// TIA Portal V19 export
FUNCTION "ALARMS" : Void   // FC16, LAD
{ S7_Optimized_Access := 'TRUE' }
// stored: SetENOAutomatically false
   VAR_TEMP   // added for the SCL form of the ladder/FBD networks
      _w1 : Bool;
   END_VAR
BEGIN

REGION Network 1: EMG ALARM
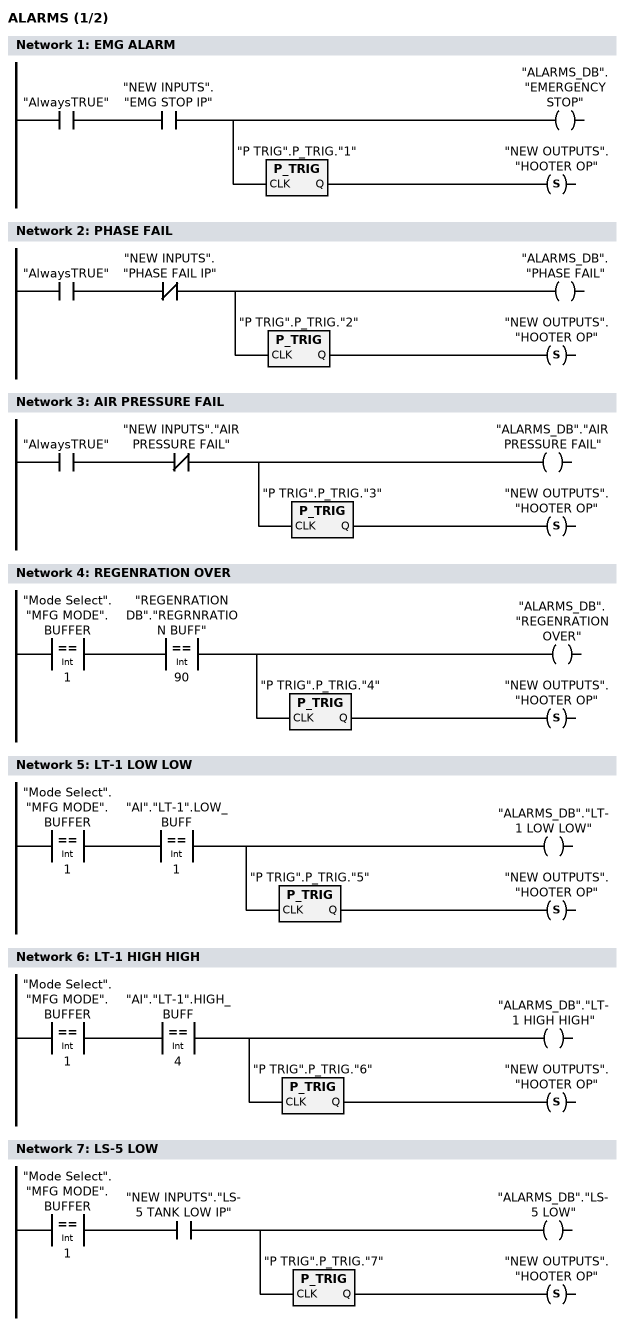
   RUNG wire#powerrail
      Contact( "AlwaysTRUE" )
      Contact( "NEW INPUTS"."EMG STOP IP" )
      wire#w1
      Coil( "ALARMS_DB"."EMERGENCY STOP" )
   END_RUNG
   RUNG wire#w1
      P_Trig( "P TRIG".P_TRIG."1" )
      S_Coil( "NEW OUTPUTS"."HOOTER OP" )
   END_RUNG
   // the same network as SCL:
   "ALARMS_DB"."EMERGENCY STOP" := "AlwaysTRUE" AND "NEW INPUTS"."EMG STOP IP";
   #_w1 := "ALARMS_DB"."EMERGENCY STOP" AND NOT "P TRIG".P_TRIG."1";   // rising edge
   "P TRIG".P_TRIG."1" := "ALARMS_DB"."EMERGENCY STOP";
   IF #_w1 THEN "NEW OUTPUTS"."HOOTER OP" := TRUE; END_IF;
END_REGION

REGION Network 2: PHASE FAIL
   RUNG wire#powerrail
      Contact( "AlwaysTRUE" )
      I_Contact( "NEW INPUTS"."PHASE FAIL IP" )
      wire#w1
      Coil( "ALARMS_DB"."PHASE FAIL" )
   END_RUNG
   RUNG wire#w1
      P_Trig( "P TRIG".P_TRIG."2" )
      S_Coil( "NEW OUTPUTS"."HOOTER OP" )
   END_RUNG
   // the same network as SCL:
   "ALARMS_DB"."PHASE FAIL" := "AlwaysTRUE" AND NOT "NEW INPUTS"."PHASE FAIL IP";
   #_w1 := "ALARMS_DB"."PHASE FAIL" AND NOT "P TRIG".P_TRIG."2";   // rising edge
   "P TRIG".P_TRIG."2" := "ALARMS_DB"."PHASE FAIL";
   IF #_w1 THEN "NEW OUTPUTS"."HOOTER OP" := TRUE; END_IF;
END_REGION

REGION Network 3: AIR PRESSURE FAIL
   RUNG wire#powerrail
      Contact( "AlwaysTRUE" )
      I_Contact( "NEW INPUTS"."AIR PRESSURE FAIL" )
      wire#w1
      Coil( "ALARMS_DB"."AIR PRESSURE FAIL" )
   END_RUNG
   RUNG wire#w1
      P_Trig( "P TRIG".P_TRIG."3" )
      S_Coil( "NEW OUTPUTS"."HOOTER OP" )
   END_RUNG
   // the same network as SCL:
   "ALARMS_DB"."AIR PRESSURE FAIL" := "AlwaysTRUE" AND NOT "NEW INPUTS"."AIR PRESSURE FAIL";
   #_w1 := "ALARMS_DB"."AIR PRESSURE FAIL" AND NOT "P TRIG".P_TRIG."3";   // rising edge
   "P TRIG".P_TRIG."3" := "ALARMS_DB"."AIR PRESSURE FAIL";
   IF #_w1 THEN "NEW OUTPUTS"."HOOTER OP" := TRUE; END_IF;
END_REGION

REGION Network 4: REGENRATION OVER
   RUNG wire#powerrail
      { S7_Templates := "SrcType := Int" } EQ_Contact(in1 := "Mode Select"."MFG MODE".BUFFER, in2 := 1)
      { S7_Templates := "SrcType := Int" } EQ_Contact(in1 := "REGENRATION DB"."REGRNRATION BUFF", in2 := 90)
      wire#w1
      Coil( "ALARMS_DB"."REGENRATION OVER" )
   END_RUNG
   RUNG wire#w1
      P_Trig( "P TRIG".P_TRIG."4" )
      S_Coil( "NEW OUTPUTS"."HOOTER OP" )
   END_RUNG
   // the same network as SCL:
   "ALARMS_DB"."REGENRATION OVER" := ("Mode Select"."MFG MODE".BUFFER = 1) AND ("REGENRATION DB"."REGRNRATION BUFF" = 90);
   #_w1 := "ALARMS_DB"."REGENRATION OVER" AND NOT "P TRIG".P_TRIG."4";   // rising edge
   "P TRIG".P_TRIG."4" := "ALARMS_DB"."REGENRATION OVER";
   IF #_w1 THEN "NEW OUTPUTS"."HOOTER OP" := TRUE; END_IF;
END_REGION

REGION Network 5: LT-1 LOW LOW
   RUNG wire#powerrail
      { S7_Templates := "SrcType := Int" } EQ_Contact(in1 := "Mode Select"."MFG MODE".BUFFER, in2 := 1)
      { S7_Templates := "SrcType := Int" } EQ_Contact(in1 := "AI"."LT-1".LOW_BUFF, in2 := 1)
      wire#w1
      Coil( "ALARMS_DB"."LT-1 LOW LOW" )
   END_RUNG
   RUNG wire#w1
      P_Trig( "P TRIG".P_TRIG."5" )
      S_Coil( "NEW OUTPUTS"."HOOTER OP" )
   END_RUNG
   // the same network as SCL:
   "ALARMS_DB"."LT-1 LOW LOW" := ("Mode Select"."MFG MODE".BUFFER = 1) AND ("AI"."LT-1".LOW_BUFF = 1);
   #_w1 := "ALARMS_DB"."LT-1 LOW LOW" AND NOT "P TRIG".P_TRIG."5";   // rising edge
   "P TRIG".P_TRIG."5" := "ALARMS_DB"."LT-1 LOW LOW";
   IF #_w1 THEN "NEW OUTPUTS"."HOOTER OP" := TRUE; END_IF;
END_REGION

REGION Network 6: LT-1 HIGH HIGH
   RUNG wire#powerrail
      { S7_Templates := "SrcType := Int" } EQ_Contact(in1 := "Mode Select"."MFG MODE".BUFFER, in2 := 1)
      { S7_Templates := "SrcType := Int" } EQ_Contact(in1 := "AI"."LT-1".HIGH_BUFF, in2 := 4)
      wire#w1
      Coil( "ALARMS_DB"."LT-1 HIGH HIGH" )
   END_RUNG
   RUNG wire#w1
      P_Trig( "P TRIG".P_TRIG."6" )
      S_Coil( "NEW OUTPUTS"."HOOTER OP" )
   END_RUNG
   // the same network as SCL:
   "ALARMS_DB"."LT-1 HIGH HIGH" := ("Mode Select"."MFG MODE".BUFFER = 1) AND ("AI"."LT-1".HIGH_BUFF = 4);
   #_w1 := "ALARMS_DB"."LT-1 HIGH HIGH" AND NOT "P TRIG".P_TRIG."6";   // rising edge
   "P TRIG".P_TRIG."6" := "ALARMS_DB"."LT-1 HIGH HIGH";
   IF #_w1 THEN "NEW OUTPUTS"."HOOTER OP" := TRUE; END_IF;
END_REGION

REGION Network 7: LS-5 LOW
   RUNG wire#powerrail
      { S7_Templates := "SrcType := Int" } EQ_Contact(in1 := "Mode Select"."MFG MODE".BUFFER, in2 := 1)
      Contact( "NEW INPUTS"."LS-5 TANK LOW IP" )
      wire#w1
      Coil( "ALARMS_DB"."LS-5 LOW" )
   END_RUNG
   RUNG wire#w1
      P_Trig( "P TRIG".P_TRIG."7" )
      S_Coil( "NEW OUTPUTS"."HOOTER OP" )
   END_RUNG
   // the same network as SCL:
   "ALARMS_DB"."LS-5 LOW" := ("Mode Select"."MFG MODE".BUFFER = 1) AND "NEW INPUTS"."LS-5 TANK LOW IP";
   #_w1 := "ALARMS_DB"."LS-5 LOW" AND NOT "P TRIG".P_TRIG."7";   // rising edge
   "P TRIG".P_TRIG."7" := "ALARMS_DB"."LS-5 LOW";
   IF #_w1 THEN "NEW OUTPUTS"."HOOTER OP" := TRUE; END_IF;
END_REGION

REGION Network 8: PS-1 LOW
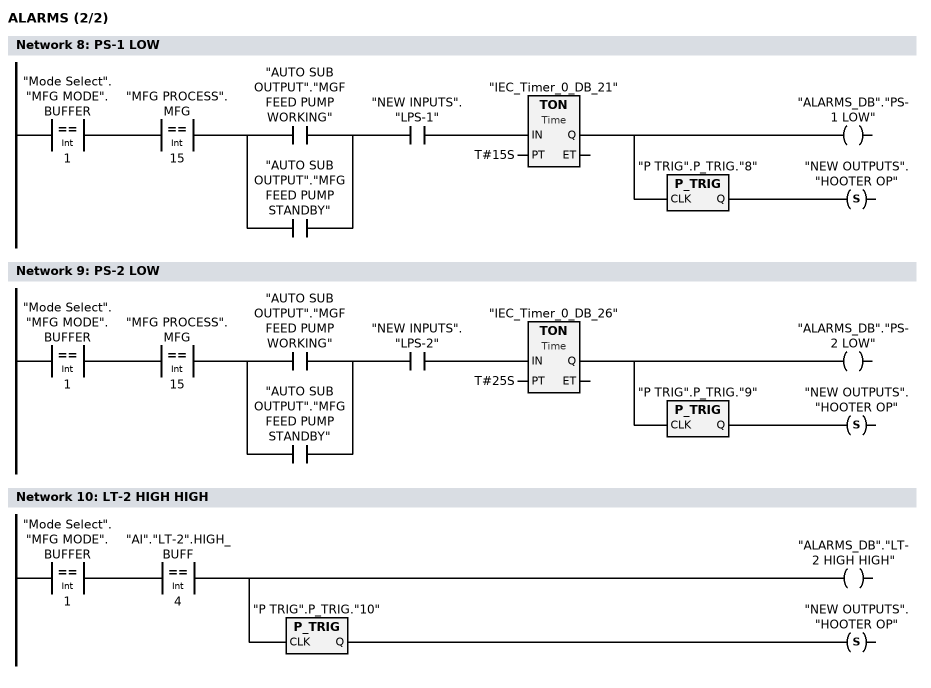
   RUNG wire#powerrail
      { S7_Templates := "SrcType := Int" } EQ_Contact(in1 := "Mode Select"."MFG MODE".BUFFER, in2 := 1)
      { S7_Templates := "SrcType := Int" } EQ_Contact(in1 := "MFG PROCESS".MFG, in2 := 15)
      wire#w1
      Contact( "AUTO SUB OUTPUT"."MGF FEED PUMP WORKING" )
      wire#w2
      Contact( "NEW INPUTS"."LPS-1" )
      { S7_Templates := "time_type := Time" } "IEC_Timer_0_DB_21".TON(pt := T#15S, et =>)
      wire#w3
      Coil( "ALARMS_DB"."PS-1 LOW" )
   END_RUNG
   RUNG wire#w1
      Contact( "AUTO SUB OUTPUT"."MFG FEED PUMP STANDBY" )
   END_RUNG wire#w2
   RUNG wire#w3
      P_Trig( "P TRIG".P_TRIG."8" )
      S_Coil( "NEW OUTPUTS"."HOOTER OP" )
   END_RUNG
   // the same network as SCL:
   "IEC_Timer_0_DB_21".TON(IN := ("Mode Select"."MFG MODE".BUFFER = 1) AND ("MFG PROCESS".MFG = 15) AND ("AUTO SUB OUTPUT"."MGF FEED PUMP WORKING" OR "AUTO SUB OUTPUT"."MFG FEED PUMP STANDBY") AND "NEW INPUTS"."LPS-1",
                           PT := T#15S);
   "ALARMS_DB"."PS-1 LOW" := "IEC_Timer_0_DB_21".Q;
   #_w1 := "IEC_Timer_0_DB_21".Q AND NOT "P TRIG".P_TRIG."8";   // rising edge
   "P TRIG".P_TRIG."8" := "IEC_Timer_0_DB_21".Q;
   IF #_w1 THEN "NEW OUTPUTS"."HOOTER OP" := TRUE; END_IF;
END_REGION

REGION Network 9: PS-2 LOW
   RUNG wire#powerrail
      { S7_Templates := "SrcType := Int" } EQ_Contact(in1 := "Mode Select"."MFG MODE".BUFFER, in2 := 1)
      { S7_Templates := "SrcType := Int" } EQ_Contact(in1 := "MFG PROCESS".MFG, in2 := 15)
      wire#w1
      Contact( "AUTO SUB OUTPUT"."MGF FEED PUMP WORKING" )
      wire#w2
      Contact( "NEW INPUTS"."LPS-2" )
      { S7_Templates := "time_type := Time" } "IEC_Timer_0_DB_26".TON(pt := T#25S, et =>)
      wire#w3
      Coil( "ALARMS_DB"."PS-2 LOW" )
   END_RUNG
   RUNG wire#w1
      Contact( "AUTO SUB OUTPUT"."MFG FEED PUMP STANDBY" )
   END_RUNG wire#w2
   RUNG wire#w3
      P_Trig( "P TRIG".P_TRIG."9" )
      S_Coil( "NEW OUTPUTS"."HOOTER OP" )
   END_RUNG
   // the same network as SCL:
   "IEC_Timer_0_DB_26".TON(IN := ("Mode Select"."MFG MODE".BUFFER = 1) AND ("MFG PROCESS".MFG = 15) AND ("AUTO SUB OUTPUT"."MGF FEED PUMP WORKING" OR "AUTO SUB OUTPUT"."MFG FEED PUMP STANDBY") AND "NEW INPUTS"."LPS-2",
                           PT := T#25S);
   "ALARMS_DB"."PS-2 LOW" := "IEC_Timer_0_DB_26".Q;
   #_w1 := "IEC_Timer_0_DB_26".Q AND NOT "P TRIG".P_TRIG."9";   // rising edge
   "P TRIG".P_TRIG."9" := "IEC_Timer_0_DB_26".Q;
   IF #_w1 THEN "NEW OUTPUTS"."HOOTER OP" := TRUE; END_IF;
END_REGION

REGION Network 10: LT-2 HIGH HIGH
   RUNG wire#powerrail
      { S7_Templates := "SrcType := Int" } EQ_Contact(in1 := "Mode Select"."MFG MODE".BUFFER, in2 := 1)
      { S7_Templates := "SrcType := Int" } EQ_Contact(in1 := "AI"."LT-2".HIGH_BUFF, in2 := 4)
      wire#w1
      Coil( "ALARMS_DB"."LT-2 HIGH HIGH" )
   END_RUNG
   RUNG wire#w1
      P_Trig( "P TRIG".P_TRIG."10" )
      S_Coil( "NEW OUTPUTS"."HOOTER OP" )
   END_RUNG
   // the same network as SCL:
   "ALARMS_DB"."LT-2 HIGH HIGH" := ("Mode Select"."MFG MODE".BUFFER = 1) AND ("AI"."LT-2".HIGH_BUFF = 4);
   #_w1 := "ALARMS_DB"."LT-2 HIGH HIGH" AND NOT "P TRIG".P_TRIG."10";   // rising edge
   "P TRIG".P_TRIG."10" := "ALARMS_DB"."LT-2 HIGH HIGH";
   IF #_w1 THEN "NEW OUTPUTS"."HOOTER OP" := TRUE; END_IF;
END_REGION
END_FUNCTION
